// TIA Portal V17 export
// export: Created 2025-05-22T12:26:37.2129325Z, ExportSetting WithDefaults, DisplayName Totally Integrated Automation Portal, DisplayVersion V17 Update 8, DisplayName TIA Portal Openness, DisplayVersion V17 Update 8, DisplayName TIA Portal Version Control Interface, DisplayVersion V17, DisplayName SINAMICS Startdrive Advanced, DisplayVersion V17 SP2, DisplayName SINAMICS Startdrive G110M, G120, G120C, G120D, G120P, G115D, DisplayVersion V17 SP2, DisplayName SINAMICS Startdrive G130, G150, S120, S150, SINAMICS MV, S210, DisplayVersion V17 SP2, DisplayName STEP 7 Professional, DisplayVersion V17 Update 8, DisplayName SINUMERIK ONE STEP 7 Toolbox, DisplayVersion V17 Update 12, DisplayName SINUMERIK ONE PLC Basic Program Plus, DisplayVersion V17 Update 12, DisplayName SINUMERIK 840D sl STEP 7 Toolbox, DisplayVersion V17 Update 12, DisplayName STEP 7 Safety, DisplayVersion V17 Update 6, DisplayName WinCC Advanced, DisplayVersion V17 Update 8
FUNCTION_BLOCK "FB2500_FIXTURE_CLADDING"   // FB2500, LAD
{ S7_Optimized_Access := 'FALSE' }
VERSION : 0.1
// stored: AutoNumber false, IsIECCheckEnabled false, SetENOAutomatically false, UDAEnableTagReadback false
   VAR_INPUT
      PART_PRESENT_FACE_SENSOR : Bool;   // PART PRESENT FACE SENSOR
      PART_STATUS_PRESENT : Bool;   // PART STATUS PRESENT
      PART_STATUS_VIRTUAL_PART : Bool;   // PART STATUS VIRTUAL PART
      PART_STATUS_MASTER_PART : Bool;   // PART STATUS MASTER PART
      STATION_PART_PRESENT : Bool;   // STATION 1 PART PRESENT IPUT
      STATION_NO_PART : Bool;   // STATION 1 NO PART
      STATION_PART_HAT_POSITION : Bool;   // STATION 1 PART PRESENT
      STATION_PART_CLAMPED : Bool;   // STATION 1 PART CLAMPED
      STATION_PART_UNCLAMPED : Bool;   // STATION 1 PART UNCLAMPED
      STATION_CLAMPED_WITHOUT_PART : Bool;   // STATION 1 CLAMPED WITHOUT PART
      VERIFY_FIXTURE_CLAMPED : Bool;   // VERIFY FIXTURE REMAINS CLAMPED
      GRIPPER_CLOSE : Bool;   // GRIPPER CLOSE ACTION
      GRIPPER_OPEN : Bool;   // GRIPPER OPEN ACTION
      GRIPPER_CLOSED : Bool;   // GRIPPER CLOSED STATUS
      "GRIPPER OPENED" : Bool;   // GRIPPER OPENED STATUS
      M_FIXTURE_GRIPPER_CLOSE : Bool;   // M CODE FIXTURE GRIPPER CLOSE
      M_FIXTURE_GRIPPER_OPEN : Bool;   // M CODE FIXTURE GRIPPER OPEN
      UP_SEALING_STRUCTURE_CLOSED : Bool;   // UP SEALING STRUCTURE CLOSED
      DOWN_SEALING_STRUCTURE_CLOSED : Bool;   // DOWN SEALING STRUCTURE CLOSED
      PART_TYPE_FIXTURES : Bool;   // PART TYPE UNIT FIXTURES
      ROBOT_PART_LOAD_UNLOAD : Bool;   // PART LOAD/UNLOAD FROM ROBOT
      ROBOT_OUT_OF_COLLISION : Bool;   // ROBOT OUT OF COLLISION MACHINE UNIT
      E_AXIS_HOME_POS : Bool;   // E AXIS IN HOME POSITION
      W_AXIS_CLAMP_CHECK_POS : Bool;   // W AXIS IN CHECK CLAMP POSITION
      W_AXIS_UNCLAMP_CHECK_POS : Bool;   // W AXIS IN CHECK UNCLAMP POSITION
      UNIT_NO : UInt;   // UNIT NUMBER
      FIXTURE_NO : UInt;   // FIXTURE NUMBER
   END_VAR
   VAR_OUTPUT
      NOT_CLAMPED_DURING_MACHINING_A : Bool;   // NOT CLAMPED DURING MACHINING ALARM
      PART_PRESENT_DISCORDANCY_A : Bool;   // PART PRESENT DISCORDANCY ALARM
      PART_TYPE_DISCORDANCY_A : Bool;   // PART TYPE DISCORDANCY ALARM
      PART_TYPE_ORIENTATED_DISCORDANCY_A : Bool;   // PART TYPE ORIENTATED DISCORDANCY ALARM
   END_VAR
   VAR DB_SPECIFIC
      DATA : "FIXTURE_STATUS";
   END_VAR
   VAR_TEMP
      DB_NUMBER : DInt;
   END_VAR
   VAR_TEMP   // added for the SCL form of the ladder/FBD networks
      _w1 : Bool;
      _w2 : Bool;
      _w3 : Bool;
      _w4 : Bool;
      _w5 : Bool;
      _w6 : Bool;
      _w7 : Bool;
      _w8 : Bool;
      _w9 : Bool;
   END_VAR
BEGIN

NETWORK
TITLE = READ INSTANCE DB
      L     DINO;
      +     10#800000;
      T     #DB_NUMBER;


REGION Network 2: FIXTURE INPUT PART A PRESENT
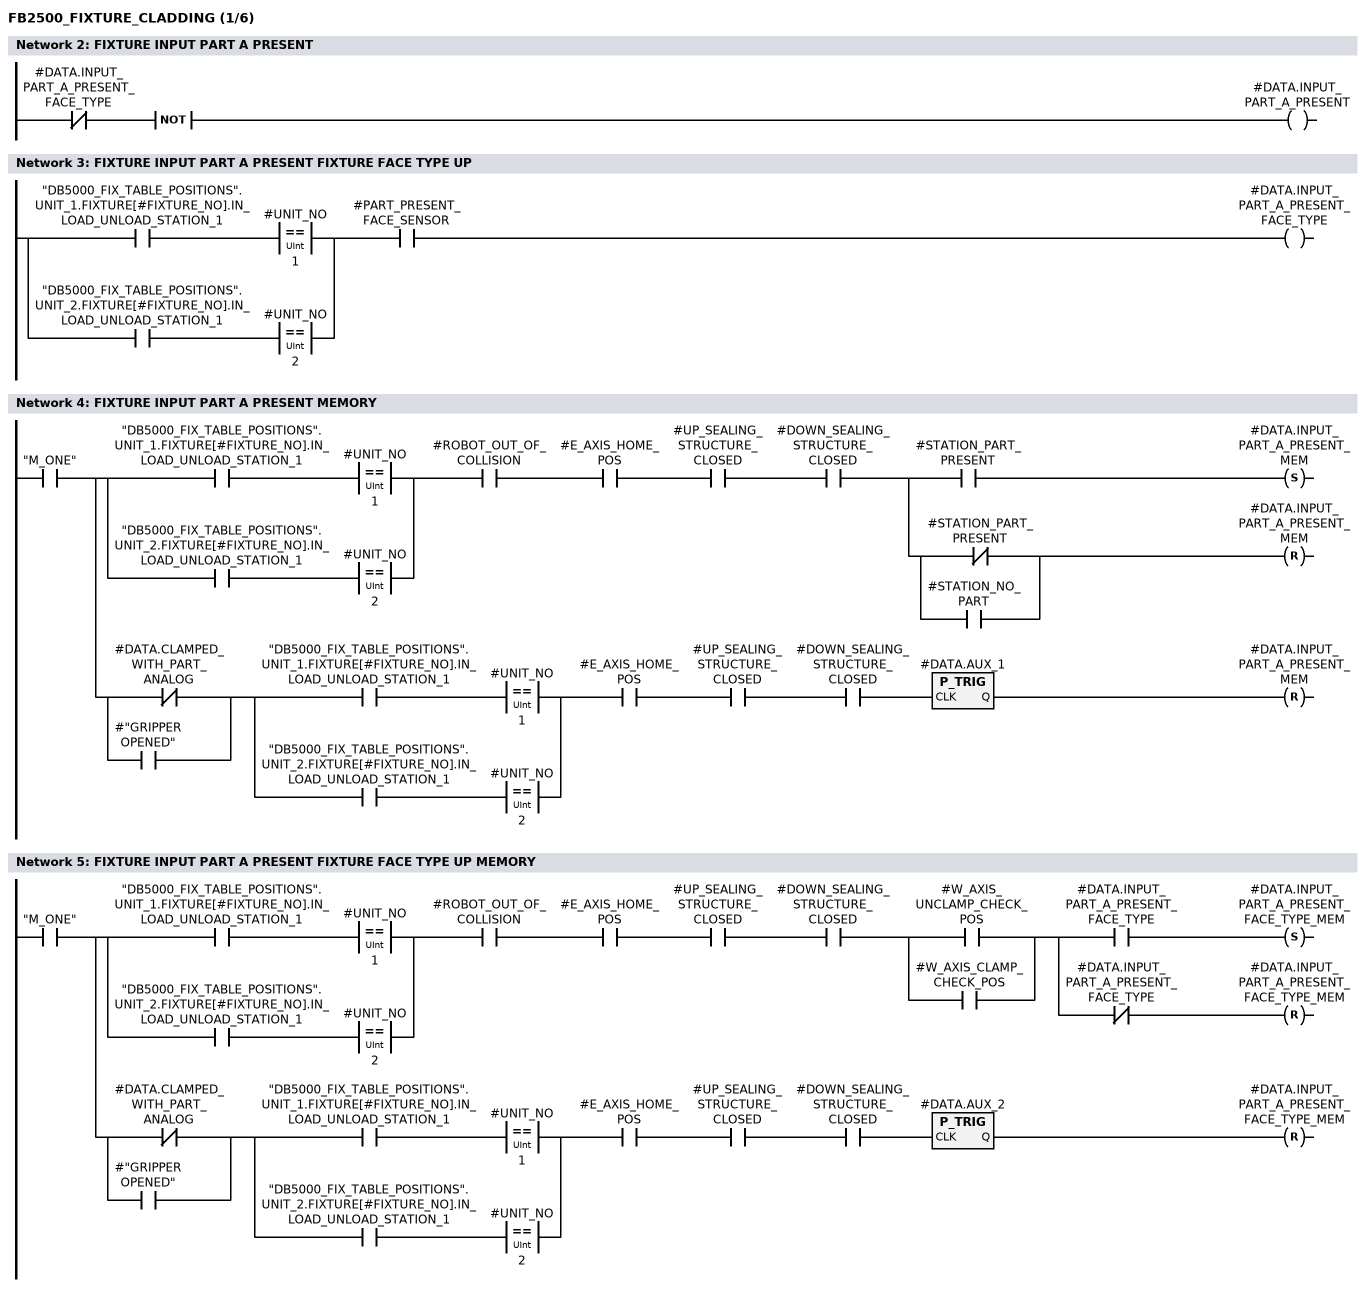
   RUNG wire#powerrail
      I_Contact( #DATA.INPUT_PART_A_PRESENT_FACE_TYPE )
      Not()
      Coil( #DATA.INPUT_PART_A_PRESENT )
   END_RUNG
   // the same network as SCL:
   #DATA.INPUT_PART_A_PRESENT := NOT (NOT #DATA.INPUT_PART_A_PRESENT_FACE_TYPE);
END_REGION

REGION Network 3: FIXTURE INPUT PART A PRESENT FIXTURE FACE TYPE UP
   RUNG wire#powerrail
      Contact( "DB5000_FIX_TABLE_POSITIONS".UNIT_1.FIXTURE[#FIXTURE_NO].IN_LOAD_UNLOAD_STATION_1 )
      { S7_Templates := "SrcType := UInt" } EQ_Contact(in1 := #UNIT_NO, in2 := 1)
      wire#w1
      Contact( #PART_PRESENT_FACE_SENSOR )
      Coil( #DATA.INPUT_PART_A_PRESENT_FACE_TYPE )
   END_RUNG
   RUNG wire#powerrail
      Contact( "DB5000_FIX_TABLE_POSITIONS".UNIT_2.FIXTURE[#FIXTURE_NO].IN_LOAD_UNLOAD_STATION_1 )
      { S7_Templates := "SrcType := UInt" } EQ_Contact(in1 := #UNIT_NO, in2 := 2)
   END_RUNG wire#w1
   // the same network as SCL:
   #DATA.INPUT_PART_A_PRESENT_FACE_TYPE := (("DB5000_FIX_TABLE_POSITIONS".UNIT_1.FIXTURE[#FIXTURE_NO].IN_LOAD_UNLOAD_STATION_1 AND (#UNIT_NO = 1)) OR ("DB5000_FIX_TABLE_POSITIONS".UNIT_2.FIXTURE[#FIXTURE_NO].IN_LOAD_UNLOAD_STATION_1 AND (#UNIT_NO = 2))) AND #PART_PRESENT_FACE_SENSOR;
END_REGION

REGION Network 4: FIXTURE INPUT PART A PRESENT MEMORY
   RUNG wire#powerrail
      Contact( "M_ONE" )
      wire#w1
      Contact( "DB5000_FIX_TABLE_POSITIONS".UNIT_1.FIXTURE[#FIXTURE_NO].IN_LOAD_UNLOAD_STATION_1 )
      { S7_Templates := "SrcType := UInt" } EQ_Contact(in1 := #UNIT_NO, in2 := 1)
      wire#w2
      Contact( #ROBOT_OUT_OF_COLLISION )
      Contact( #E_AXIS_HOME_POS )
      Contact( #UP_SEALING_STRUCTURE_CLOSED )
      Contact( #DOWN_SEALING_STRUCTURE_CLOSED )
      wire#w3
      Contact( #STATION_PART_PRESENT )
      S_Coil( #DATA.INPUT_PART_A_PRESENT_MEM )
   END_RUNG
   RUNG wire#w1
      Contact( "DB5000_FIX_TABLE_POSITIONS".UNIT_2.FIXTURE[#FIXTURE_NO].IN_LOAD_UNLOAD_STATION_1 )
      { S7_Templates := "SrcType := UInt" } EQ_Contact(in1 := #UNIT_NO, in2 := 2)
   END_RUNG wire#w2
   RUNG wire#w3
      I_Contact( #STATION_PART_PRESENT )
      wire#w4
      R_Coil( #DATA.INPUT_PART_A_PRESENT_MEM )
   END_RUNG
   RUNG wire#w3
      Contact( #STATION_NO_PART )
   END_RUNG wire#w4
   RUNG wire#w1
      I_Contact( #DATA.CLAMPED_WITH_PART_ANALOG )
      wire#w5
      Contact( "DB5000_FIX_TABLE_POSITIONS".UNIT_1.FIXTURE[#FIXTURE_NO].IN_LOAD_UNLOAD_STATION_1 )
      { S7_Templates := "SrcType := UInt" } EQ_Contact(in1 := #UNIT_NO, in2 := 1)
      wire#w6
      Contact( #E_AXIS_HOME_POS )
      Contact( #UP_SEALING_STRUCTURE_CLOSED )
      Contact( #DOWN_SEALING_STRUCTURE_CLOSED )
      P_Trig( #DATA.AUX_1 )
      R_Coil( #DATA.INPUT_PART_A_PRESENT_MEM )
   END_RUNG
   RUNG wire#w1
      Contact( #"GRIPPER OPENED" )
   END_RUNG wire#w5
   RUNG wire#w5
      Contact( "DB5000_FIX_TABLE_POSITIONS".UNIT_2.FIXTURE[#FIXTURE_NO].IN_LOAD_UNLOAD_STATION_1 )
      { S7_Templates := "SrcType := UInt" } EQ_Contact(in1 := #UNIT_NO, in2 := 2)
   END_RUNG wire#w6
   // the same network as SCL:
   #_w1 := "M_ONE" AND (("DB5000_FIX_TABLE_POSITIONS".UNIT_1.FIXTURE[#FIXTURE_NO].IN_LOAD_UNLOAD_STATION_1 AND (#UNIT_NO = 1)) OR ("DB5000_FIX_TABLE_POSITIONS".UNIT_2.FIXTURE[#FIXTURE_NO].IN_LOAD_UNLOAD_STATION_1 AND (#UNIT_NO = 2))) AND #ROBOT_OUT_OF_COLLISION AND #E_AXIS_HOME_POS AND #UP_SEALING_STRUCTURE_CLOSED AND #DOWN_SEALING_STRUCTURE_CLOSED;
   IF #_w1 AND #STATION_PART_PRESENT THEN #DATA.INPUT_PART_A_PRESENT_MEM := TRUE; END_IF;
   IF #_w1 AND (NOT #STATION_PART_PRESENT OR #STATION_NO_PART) THEN
       #DATA.INPUT_PART_A_PRESENT_MEM := FALSE;
   END_IF;
   #_w2 := "M_ONE" AND (NOT #DATA.CLAMPED_WITH_PART_ANALOG OR #"GRIPPER OPENED") AND (("DB5000_FIX_TABLE_POSITIONS".UNIT_1.FIXTURE[#FIXTURE_NO].IN_LOAD_UNLOAD_STATION_1 AND (#UNIT_NO = 1)) OR ("DB5000_FIX_TABLE_POSITIONS".UNIT_2.FIXTURE[#FIXTURE_NO].IN_LOAD_UNLOAD_STATION_1 AND (#UNIT_NO = 2))) AND #E_AXIS_HOME_POS AND #UP_SEALING_STRUCTURE_CLOSED AND #DOWN_SEALING_STRUCTURE_CLOSED;
   #_w3 := #_w2 AND NOT #DATA.AUX_1;   // rising edge
   #DATA.AUX_1 := #_w2;
   IF #_w3 THEN #DATA.INPUT_PART_A_PRESENT_MEM := FALSE; END_IF;
END_REGION

REGION Network 5: FIXTURE INPUT PART A PRESENT FIXTURE FACE TYPE UP MEMORY
   RUNG wire#powerrail
      Contact( "M_ONE" )
      wire#w1
      Contact( "DB5000_FIX_TABLE_POSITIONS".UNIT_1.FIXTURE[#FIXTURE_NO].IN_LOAD_UNLOAD_STATION_1 )
      { S7_Templates := "SrcType := UInt" } EQ_Contact(in1 := #UNIT_NO, in2 := 1)
      wire#w2
      Contact( #ROBOT_OUT_OF_COLLISION )
      Contact( #E_AXIS_HOME_POS )
      Contact( #UP_SEALING_STRUCTURE_CLOSED )
      Contact( #DOWN_SEALING_STRUCTURE_CLOSED )
      wire#w3
      Contact( #W_AXIS_UNCLAMP_CHECK_POS )
      wire#w4
      Contact( #DATA.INPUT_PART_A_PRESENT_FACE_TYPE )
      S_Coil( #DATA.INPUT_PART_A_PRESENT_FACE_TYPE_MEM )
   END_RUNG
   RUNG wire#w1
      Contact( "DB5000_FIX_TABLE_POSITIONS".UNIT_2.FIXTURE[#FIXTURE_NO].IN_LOAD_UNLOAD_STATION_1 )
      { S7_Templates := "SrcType := UInt" } EQ_Contact(in1 := #UNIT_NO, in2 := 2)
   END_RUNG wire#w2
   RUNG wire#w3
      Contact( #W_AXIS_CLAMP_CHECK_POS )
   END_RUNG wire#w4
   RUNG wire#w4
      I_Contact( #DATA.INPUT_PART_A_PRESENT_FACE_TYPE )
      R_Coil( #DATA.INPUT_PART_A_PRESENT_FACE_TYPE_MEM )
   END_RUNG
   RUNG wire#w1
      I_Contact( #DATA.CLAMPED_WITH_PART_ANALOG )
      wire#w5
      Contact( "DB5000_FIX_TABLE_POSITIONS".UNIT_1.FIXTURE[#FIXTURE_NO].IN_LOAD_UNLOAD_STATION_1 )
      { S7_Templates := "SrcType := UInt" } EQ_Contact(in1 := #UNIT_NO, in2 := 1)
      wire#w6
      Contact( #E_AXIS_HOME_POS )
      Contact( #UP_SEALING_STRUCTURE_CLOSED )
      Contact( #DOWN_SEALING_STRUCTURE_CLOSED )
      P_Trig( #DATA.AUX_2 )
      R_Coil( #DATA.INPUT_PART_A_PRESENT_FACE_TYPE_MEM )
   END_RUNG
   RUNG wire#w1
      Contact( #"GRIPPER OPENED" )
   END_RUNG wire#w5
   RUNG wire#w5
      Contact( "DB5000_FIX_TABLE_POSITIONS".UNIT_2.FIXTURE[#FIXTURE_NO].IN_LOAD_UNLOAD_STATION_1 )
      { S7_Templates := "SrcType := UInt" } EQ_Contact(in1 := #UNIT_NO, in2 := 2)
   END_RUNG wire#w6
   // the same network as SCL:
   #_w1 := "M_ONE" AND (("DB5000_FIX_TABLE_POSITIONS".UNIT_1.FIXTURE[#FIXTURE_NO].IN_LOAD_UNLOAD_STATION_1 AND (#UNIT_NO = 1)) OR ("DB5000_FIX_TABLE_POSITIONS".UNIT_2.FIXTURE[#FIXTURE_NO].IN_LOAD_UNLOAD_STATION_1 AND (#UNIT_NO = 2))) AND #ROBOT_OUT_OF_COLLISION AND #E_AXIS_HOME_POS AND #UP_SEALING_STRUCTURE_CLOSED AND #DOWN_SEALING_STRUCTURE_CLOSED AND (#W_AXIS_UNCLAMP_CHECK_POS OR #W_AXIS_CLAMP_CHECK_POS);
   IF #_w1 AND #DATA.INPUT_PART_A_PRESENT_FACE_TYPE THEN
       #DATA.INPUT_PART_A_PRESENT_FACE_TYPE_MEM := TRUE;
   END_IF;
   IF #_w1 AND NOT #DATA.INPUT_PART_A_PRESENT_FACE_TYPE THEN
       #DATA.INPUT_PART_A_PRESENT_FACE_TYPE_MEM := FALSE;
   END_IF;
   #_w2 := "M_ONE" AND (NOT #DATA.CLAMPED_WITH_PART_ANALOG OR #"GRIPPER OPENED") AND (("DB5000_FIX_TABLE_POSITIONS".UNIT_1.FIXTURE[#FIXTURE_NO].IN_LOAD_UNLOAD_STATION_1 AND (#UNIT_NO = 1)) OR ("DB5000_FIX_TABLE_POSITIONS".UNIT_2.FIXTURE[#FIXTURE_NO].IN_LOAD_UNLOAD_STATION_1 AND (#UNIT_NO = 2))) AND #E_AXIS_HOME_POS AND #UP_SEALING_STRUCTURE_CLOSED AND #DOWN_SEALING_STRUCTURE_CLOSED;
   #_w3 := #_w2 AND NOT #DATA.AUX_2;   // rising edge
   #DATA.AUX_2 := #_w2;
   IF #_w3 THEN #DATA.INPUT_PART_A_PRESENT_FACE_TYPE_MEM := FALSE; END_IF;
END_REGION

REGION Network 6: ANY PART PRESENT
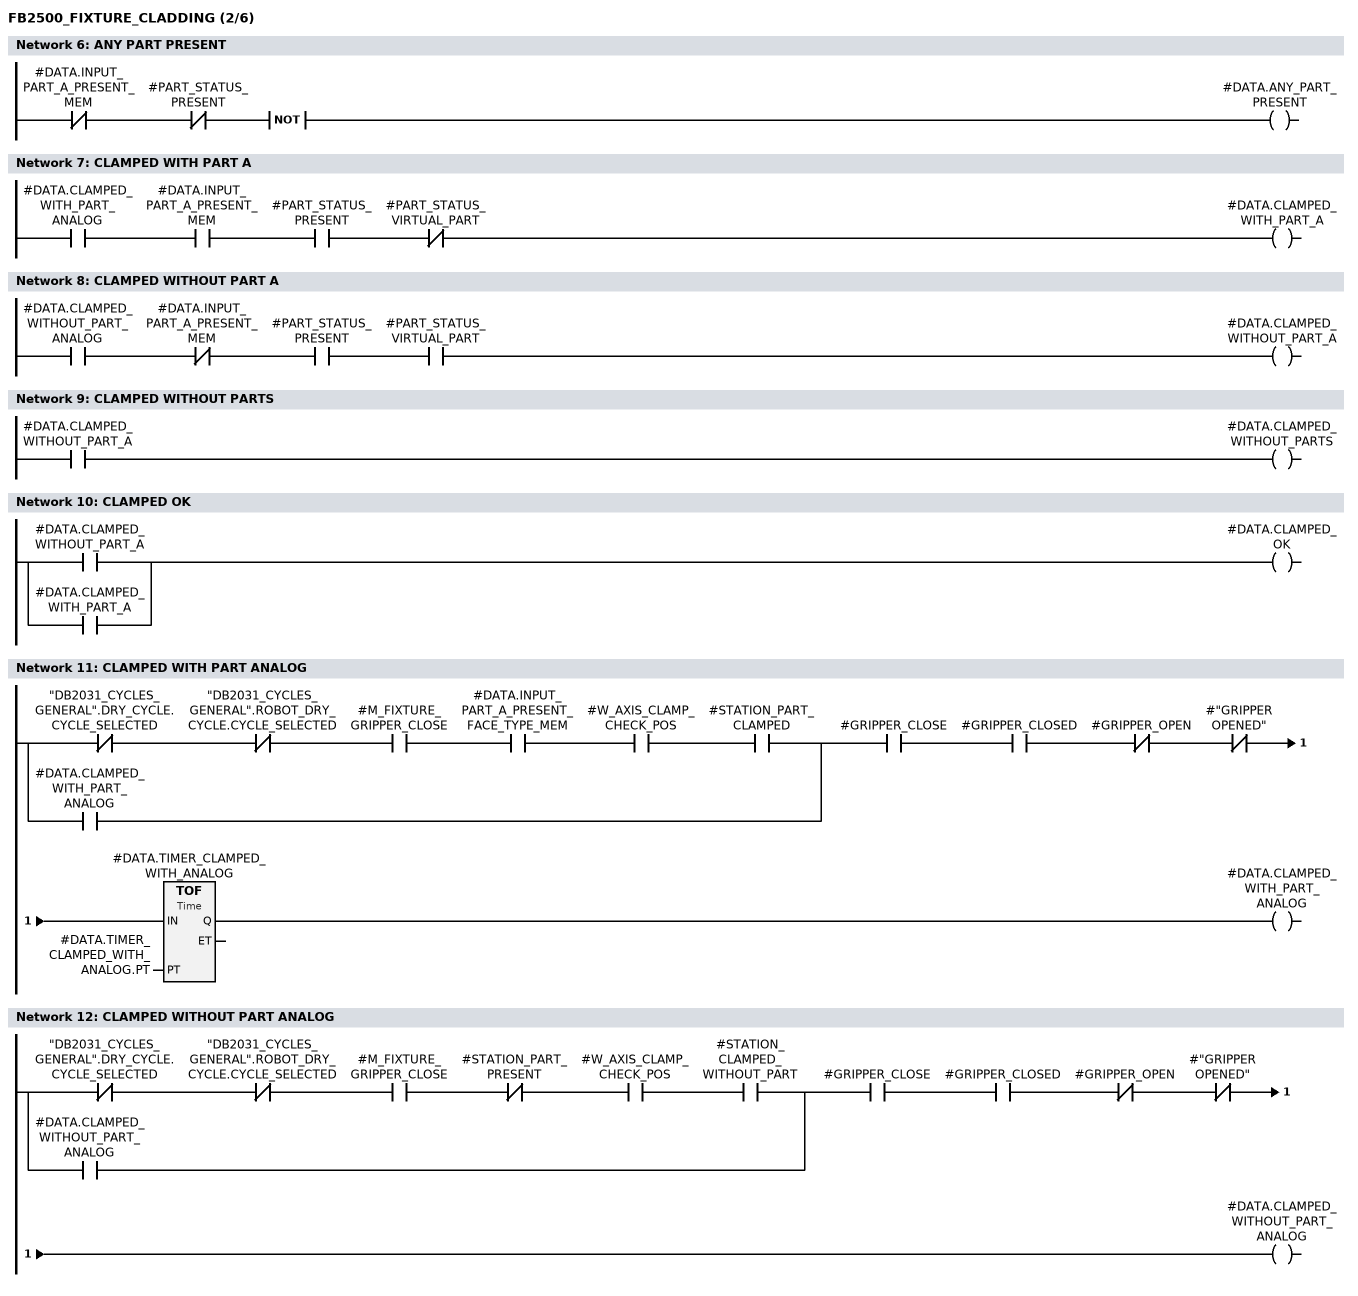
   RUNG wire#powerrail
      I_Contact( #DATA.INPUT_PART_A_PRESENT_MEM )
      I_Contact( #PART_STATUS_PRESENT )
      Not()
      Coil( #DATA.ANY_PART_PRESENT )
   END_RUNG
   // the same network as SCL:
   #DATA.ANY_PART_PRESENT := NOT (NOT #DATA.INPUT_PART_A_PRESENT_MEM AND NOT #PART_STATUS_PRESENT);
END_REGION

REGION Network 7: CLAMPED WITH PART A
   RUNG wire#powerrail
      Contact( #DATA.CLAMPED_WITH_PART_ANALOG )
      Contact( #DATA.INPUT_PART_A_PRESENT_MEM )
      Contact( #PART_STATUS_PRESENT )
      I_Contact( #PART_STATUS_VIRTUAL_PART )
      Coil( #DATA.CLAMPED_WITH_PART_A )
   END_RUNG
   // the same network as SCL:
   #DATA.CLAMPED_WITH_PART_A := #DATA.CLAMPED_WITH_PART_ANALOG AND #DATA.INPUT_PART_A_PRESENT_MEM AND #PART_STATUS_PRESENT AND NOT #PART_STATUS_VIRTUAL_PART;
END_REGION

REGION Network 8: CLAMPED WITHOUT PART A
   RUNG wire#powerrail
      Contact( #DATA.CLAMPED_WITHOUT_PART_ANALOG )
      I_Contact( #DATA.INPUT_PART_A_PRESENT_MEM )
      Contact( #PART_STATUS_PRESENT )
      Contact( #PART_STATUS_VIRTUAL_PART )
      Coil( #DATA.CLAMPED_WITHOUT_PART_A )
   END_RUNG
   // the same network as SCL:
   #DATA.CLAMPED_WITHOUT_PART_A := #DATA.CLAMPED_WITHOUT_PART_ANALOG AND NOT #DATA.INPUT_PART_A_PRESENT_MEM AND #PART_STATUS_PRESENT AND #PART_STATUS_VIRTUAL_PART;
END_REGION

REGION Network 9: CLAMPED WITHOUT PARTS
   RUNG wire#powerrail
      Contact( #DATA.CLAMPED_WITHOUT_PART_A )
      Coil( #DATA.CLAMPED_WITHOUT_PARTS )
   END_RUNG
   // the same network as SCL:
   #DATA.CLAMPED_WITHOUT_PARTS := #DATA.CLAMPED_WITHOUT_PART_A;
END_REGION

REGION Network 10: CLAMPED OK
   RUNG wire#powerrail
      Contact( #DATA.CLAMPED_WITHOUT_PART_A )
      wire#w1
      Coil( #DATA.CLAMPED_OK )
   END_RUNG
   RUNG wire#powerrail
      Contact( #DATA.CLAMPED_WITH_PART_A )
   END_RUNG wire#w1
   // the same network as SCL:
   #DATA.CLAMPED_OK := #DATA.CLAMPED_WITHOUT_PART_A OR #DATA.CLAMPED_WITH_PART_A;
END_REGION

REGION Network 11: CLAMPED WITH PART ANALOG
   RUNG wire#powerrail
      I_Contact( "DB2031_CYCLES_GENERAL".DRY_CYCLE.CYCLE_SELECTED )
      I_Contact( "DB2031_CYCLES_GENERAL".ROBOT_DRY_CYCLE.CYCLE_SELECTED )
      Contact( #M_FIXTURE_GRIPPER_CLOSE )
      Contact( #DATA.INPUT_PART_A_PRESENT_FACE_TYPE_MEM )
      Contact( #W_AXIS_CLAMP_CHECK_POS )
      Contact( #STATION_PART_CLAMPED )
      wire#w1
      Contact( #GRIPPER_CLOSE )
      Contact( #GRIPPER_CLOSED )
      I_Contact( #GRIPPER_OPEN )
      I_Contact( #"GRIPPER OPENED" )
      { S7_Templates := "time_type := Time" } #DATA.TIMER_CLAMPED_WITH_ANALOG.TOF(pt := #DATA.TIMER_CLAMPED_WITH_ANALOG.PT, et =>)
      Coil( #DATA.CLAMPED_WITH_PART_ANALOG )
   END_RUNG
   RUNG wire#powerrail
      Contact( #DATA.CLAMPED_WITH_PART_ANALOG )
   END_RUNG wire#w1
   // the same network as SCL:
   #DATA.TIMER_CLAMPED_WITH_ANALOG.TOF(IN := ((NOT "DB2031_CYCLES_GENERAL".DRY_CYCLE.CYCLE_SELECTED AND NOT "DB2031_CYCLES_GENERAL".ROBOT_DRY_CYCLE.CYCLE_SELECTED AND #M_FIXTURE_GRIPPER_CLOSE AND #DATA.INPUT_PART_A_PRESENT_FACE_TYPE_MEM AND #W_AXIS_CLAMP_CHECK_POS AND #STATION_PART_CLAMPED) OR #DATA.CLAMPED_WITH_PART_ANALOG) AND #GRIPPER_CLOSE AND #GRIPPER_CLOSED AND NOT #GRIPPER_OPEN AND NOT #"GRIPPER OPENED",
                           PT := #DATA.TIMER_CLAMPED_WITH_ANALOG.PT);
   #DATA.CLAMPED_WITH_PART_ANALOG := #DATA.TIMER_CLAMPED_WITH_ANALOG.Q;
END_REGION

REGION Network 12: CLAMPED WITHOUT PART ANALOG
   RUNG wire#powerrail
      I_Contact( "DB2031_CYCLES_GENERAL".DRY_CYCLE.CYCLE_SELECTED )
      I_Contact( "DB2031_CYCLES_GENERAL".ROBOT_DRY_CYCLE.CYCLE_SELECTED )
      Contact( #M_FIXTURE_GRIPPER_CLOSE )
      I_Contact( #STATION_PART_PRESENT )
      Contact( #W_AXIS_CLAMP_CHECK_POS )
      Contact( #STATION_CLAMPED_WITHOUT_PART )
      wire#w1
      Contact( #GRIPPER_CLOSE )
      Contact( #GRIPPER_CLOSED )
      I_Contact( #GRIPPER_OPEN )
      I_Contact( #"GRIPPER OPENED" )
      Coil( #DATA.CLAMPED_WITHOUT_PART_ANALOG )
   END_RUNG
   RUNG wire#powerrail
      Contact( #DATA.CLAMPED_WITHOUT_PART_ANALOG )
   END_RUNG wire#w1
   // the same network as SCL:
   #DATA.CLAMPED_WITHOUT_PART_ANALOG := ((NOT "DB2031_CYCLES_GENERAL".DRY_CYCLE.CYCLE_SELECTED AND NOT "DB2031_CYCLES_GENERAL".ROBOT_DRY_CYCLE.CYCLE_SELECTED AND #M_FIXTURE_GRIPPER_CLOSE AND NOT #STATION_PART_PRESENT AND #W_AXIS_CLAMP_CHECK_POS AND #STATION_CLAMPED_WITHOUT_PART) OR #DATA.CLAMPED_WITHOUT_PART_ANALOG) AND #GRIPPER_CLOSE AND #GRIPPER_CLOSED AND NOT #GRIPPER_OPEN AND NOT #"GRIPPER OPENED";
END_REGION

REGION Network 13: UNCLAMPED ANALOG
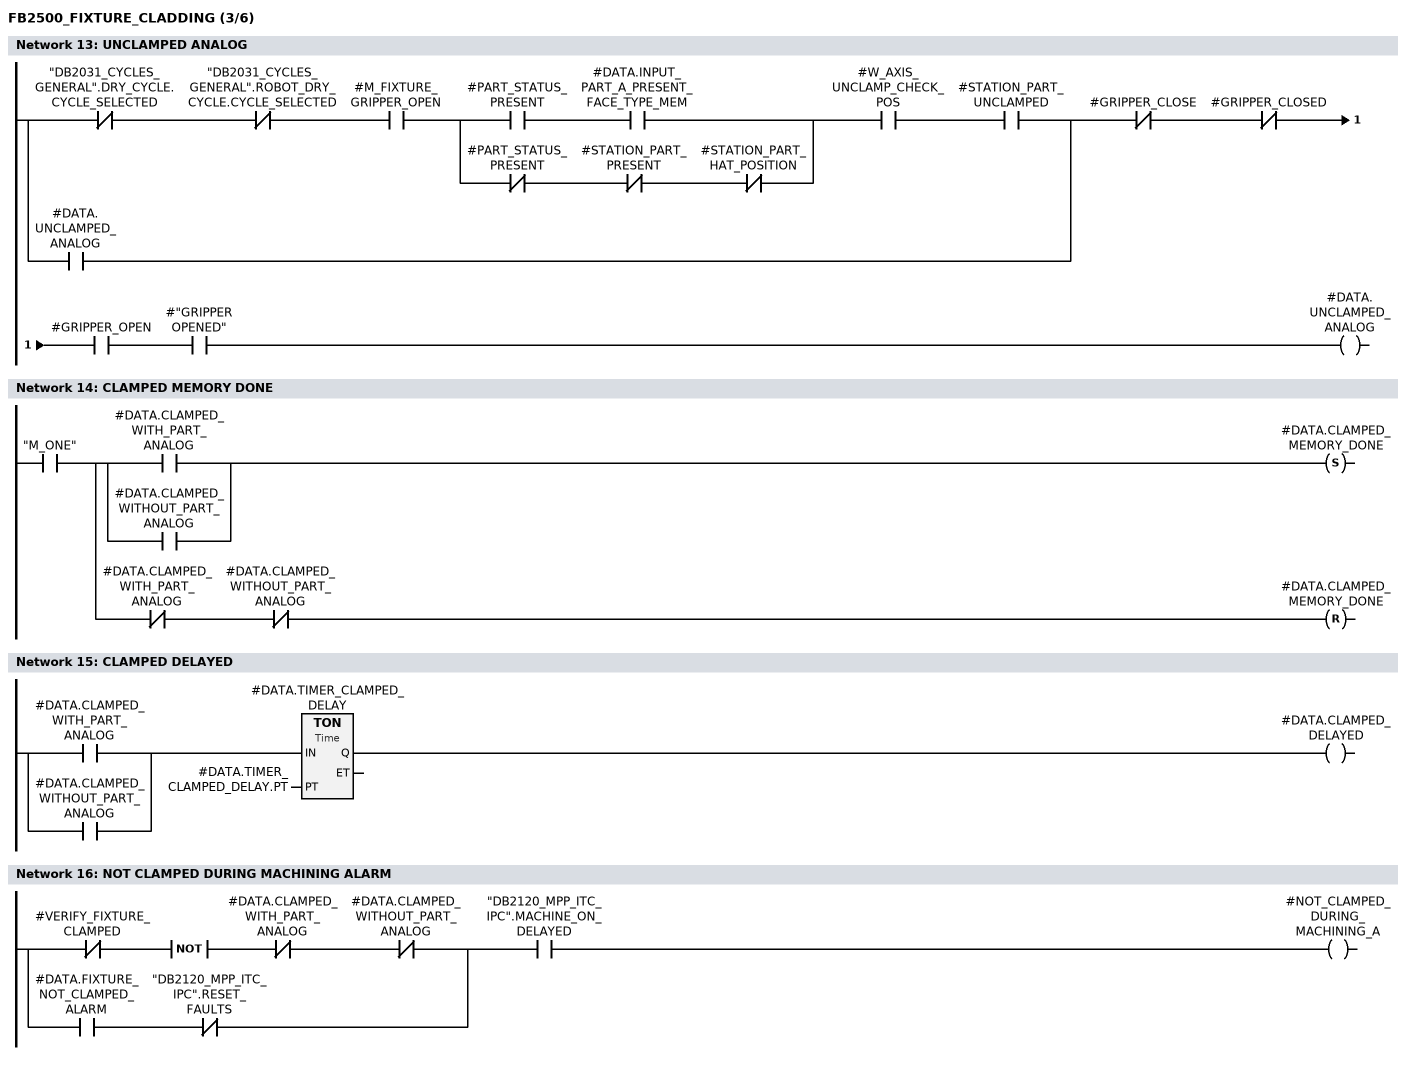
   RUNG wire#powerrail
      I_Contact( "DB2031_CYCLES_GENERAL".DRY_CYCLE.CYCLE_SELECTED )
      I_Contact( "DB2031_CYCLES_GENERAL".ROBOT_DRY_CYCLE.CYCLE_SELECTED )
      Contact( #M_FIXTURE_GRIPPER_OPEN )
      wire#w1
      Contact( #PART_STATUS_PRESENT )
      Contact( #DATA.INPUT_PART_A_PRESENT_FACE_TYPE_MEM )
      wire#w2
      Contact( #W_AXIS_UNCLAMP_CHECK_POS )
      Contact( #STATION_PART_UNCLAMPED )
      wire#w3
      I_Contact( #GRIPPER_CLOSE )
      I_Contact( #GRIPPER_CLOSED )
      Contact( #GRIPPER_OPEN )
      Contact( #"GRIPPER OPENED" )
      Coil( #DATA.UNCLAMPED_ANALOG )
   END_RUNG
   RUNG wire#w1
      I_Contact( #PART_STATUS_PRESENT )
      I_Contact( #STATION_PART_PRESENT )
      I_Contact( #STATION_PART_HAT_POSITION )
   END_RUNG wire#w2
   RUNG wire#powerrail
      Contact( #DATA.UNCLAMPED_ANALOG )
   END_RUNG wire#w3
   // the same network as SCL:
   #DATA.UNCLAMPED_ANALOG := ((NOT "DB2031_CYCLES_GENERAL".DRY_CYCLE.CYCLE_SELECTED AND NOT "DB2031_CYCLES_GENERAL".ROBOT_DRY_CYCLE.CYCLE_SELECTED AND #M_FIXTURE_GRIPPER_OPEN AND ((#PART_STATUS_PRESENT AND #DATA.INPUT_PART_A_PRESENT_FACE_TYPE_MEM) OR (NOT #PART_STATUS_PRESENT AND NOT #STATION_PART_PRESENT AND NOT #STATION_PART_HAT_POSITION)) AND #W_AXIS_UNCLAMP_CHECK_POS AND #STATION_PART_UNCLAMPED) OR #DATA.UNCLAMPED_ANALOG) AND NOT #GRIPPER_CLOSE AND NOT #GRIPPER_CLOSED AND #GRIPPER_OPEN AND #"GRIPPER OPENED";
END_REGION

REGION Network 14: CLAMPED MEMORY DONE
   RUNG wire#powerrail
      Contact( "M_ONE" )
      wire#w1
      Contact( #DATA.CLAMPED_WITH_PART_ANALOG )
      wire#w2
      S_Coil( #DATA.CLAMPED_MEMORY_DONE )
   END_RUNG
   RUNG wire#w1
      Contact( #DATA.CLAMPED_WITHOUT_PART_ANALOG )
   END_RUNG wire#w2
   RUNG wire#w1
      I_Contact( #DATA.CLAMPED_WITH_PART_ANALOG )
      I_Contact( #DATA.CLAMPED_WITHOUT_PART_ANALOG )
      R_Coil( #DATA.CLAMPED_MEMORY_DONE )
   END_RUNG
   // the same network as SCL:
   IF "M_ONE" AND (#DATA.CLAMPED_WITH_PART_ANALOG OR #DATA.CLAMPED_WITHOUT_PART_ANALOG) THEN
       #DATA.CLAMPED_MEMORY_DONE := TRUE;
   END_IF;
   IF "M_ONE" AND NOT #DATA.CLAMPED_WITH_PART_ANALOG AND NOT #DATA.CLAMPED_WITHOUT_PART_ANALOG THEN
       #DATA.CLAMPED_MEMORY_DONE := FALSE;
   END_IF;
END_REGION

REGION Network 15: CLAMPED DELAYED
   RUNG wire#powerrail
      Contact( #DATA.CLAMPED_WITH_PART_ANALOG )
      wire#w1
      { S7_Templates := "time_type := Time" } #DATA.TIMER_CLAMPED_DELAY.TON(pt := #DATA.TIMER_CLAMPED_DELAY.PT, et =>)
      Coil( #DATA.CLAMPED_DELAYED )
   END_RUNG
   RUNG wire#powerrail
      Contact( #DATA.CLAMPED_WITHOUT_PART_ANALOG )
   END_RUNG wire#w1
   // the same network as SCL:
   #DATA.TIMER_CLAMPED_DELAY.TON(IN := #DATA.CLAMPED_WITH_PART_ANALOG OR #DATA.CLAMPED_WITHOUT_PART_ANALOG,
                           PT := #DATA.TIMER_CLAMPED_DELAY.PT);
   #DATA.CLAMPED_DELAYED := #DATA.TIMER_CLAMPED_DELAY.Q;
END_REGION

REGION Network 16: NOT CLAMPED DURING MACHINING ALARM
   RUNG wire#powerrail
      I_Contact( #VERIFY_FIXTURE_CLAMPED )
      Not()
      I_Contact( #DATA.CLAMPED_WITH_PART_ANALOG )
      I_Contact( #DATA.CLAMPED_WITHOUT_PART_ANALOG )
      wire#w1
      Contact( "DB2120_MPP_ITC_IPC".MACHINE_ON_DELAYED )
      Coil( #NOT_CLAMPED_DURING_MACHINING_A )
   END_RUNG
   RUNG wire#powerrail
      Contact( #DATA.FIXTURE_NOT_CLAMPED_ALARM )
      I_Contact( "DB2120_MPP_ITC_IPC".RESET_FAULTS )
   END_RUNG wire#w1
   // the same network as SCL:
   #NOT_CLAMPED_DURING_MACHINING_A := ((NOT (NOT #VERIFY_FIXTURE_CLAMPED) AND NOT #DATA.CLAMPED_WITH_PART_ANALOG AND NOT #DATA.CLAMPED_WITHOUT_PART_ANALOG) OR (#DATA.FIXTURE_NOT_CLAMPED_ALARM AND NOT "DB2120_MPP_ITC_IPC".RESET_FAULTS)) AND "DB2120_MPP_ITC_IPC".MACHINE_ON_DELAYED;
END_REGION

REGION Network 17: PART A PRESENT DISCORDANCY ALARM
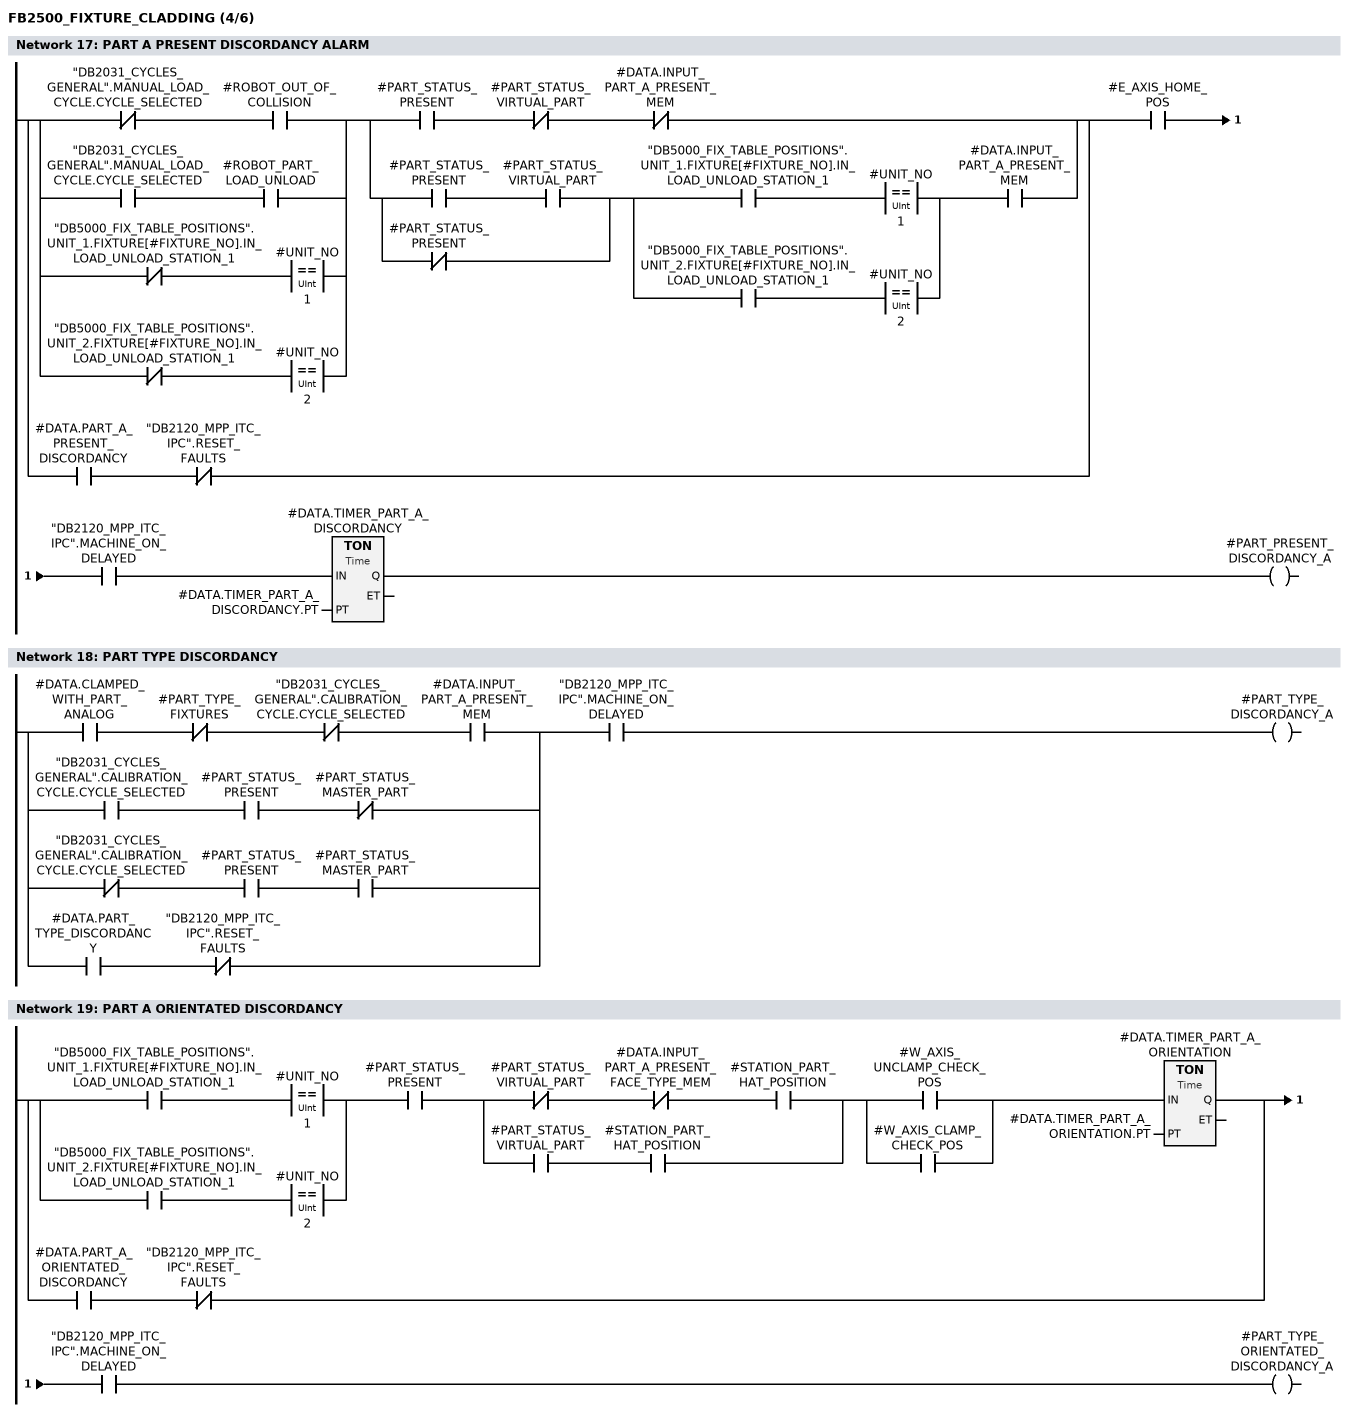
   RUNG wire#powerrail
      I_Contact( "DB2031_CYCLES_GENERAL".MANUAL_LOAD_CYCLE.CYCLE_SELECTED )
      Contact( #ROBOT_OUT_OF_COLLISION )
      wire#w1
      Contact( #PART_STATUS_PRESENT )
      I_Contact( #PART_STATUS_VIRTUAL_PART )
      I_Contact( #DATA.INPUT_PART_A_PRESENT_MEM )
      wire#w2
      Contact( #E_AXIS_HOME_POS )
      Contact( "DB2120_MPP_ITC_IPC".MACHINE_ON_DELAYED )
      { S7_Templates := "time_type := Time" } #DATA.TIMER_PART_A_DISCORDANCY.TON(pt := #DATA.TIMER_PART_A_DISCORDANCY.PT, et =>)
      Coil( #PART_PRESENT_DISCORDANCY_A )
   END_RUNG
   RUNG wire#powerrail
      Contact( "DB2031_CYCLES_GENERAL".MANUAL_LOAD_CYCLE.CYCLE_SELECTED )
      Contact( #ROBOT_PART_LOAD_UNLOAD )
   END_RUNG wire#w1
   RUNG wire#powerrail
      I_Contact( "DB5000_FIX_TABLE_POSITIONS".UNIT_1.FIXTURE[#FIXTURE_NO].IN_LOAD_UNLOAD_STATION_1 )
      { S7_Templates := "SrcType := UInt" } EQ_Contact(in1 := #UNIT_NO, in2 := 1)
   END_RUNG wire#w1
   RUNG wire#powerrail
      I_Contact( "DB5000_FIX_TABLE_POSITIONS".UNIT_2.FIXTURE[#FIXTURE_NO].IN_LOAD_UNLOAD_STATION_1 )
      { S7_Templates := "SrcType := UInt" } EQ_Contact(in1 := #UNIT_NO, in2 := 2)
   END_RUNG wire#w1
   RUNG wire#w1
      Contact( #PART_STATUS_PRESENT )
      Contact( #PART_STATUS_VIRTUAL_PART )
      wire#w3
      Contact( "DB5000_FIX_TABLE_POSITIONS".UNIT_1.FIXTURE[#FIXTURE_NO].IN_LOAD_UNLOAD_STATION_1 )
      { S7_Templates := "SrcType := UInt" } EQ_Contact(in1 := #UNIT_NO, in2 := 1)
      wire#w4
      Contact( #DATA.INPUT_PART_A_PRESENT_MEM )
   END_RUNG wire#w2
   RUNG wire#w1
      I_Contact( #PART_STATUS_PRESENT )
   END_RUNG wire#w3
   RUNG wire#w3
      Contact( "DB5000_FIX_TABLE_POSITIONS".UNIT_2.FIXTURE[#FIXTURE_NO].IN_LOAD_UNLOAD_STATION_1 )
      { S7_Templates := "SrcType := UInt" } EQ_Contact(in1 := #UNIT_NO, in2 := 2)
   END_RUNG wire#w4
   RUNG wire#powerrail
      Contact( #DATA.PART_A_PRESENT_DISCORDANCY )
      I_Contact( "DB2120_MPP_ITC_IPC".RESET_FAULTS )
   END_RUNG wire#w2
   // the same network as SCL:
   #DATA.TIMER_PART_A_DISCORDANCY.TON(IN := ((((NOT "DB2031_CYCLES_GENERAL".MANUAL_LOAD_CYCLE.CYCLE_SELECTED AND #ROBOT_OUT_OF_COLLISION) OR ("DB2031_CYCLES_GENERAL".MANUAL_LOAD_CYCLE.CYCLE_SELECTED AND #ROBOT_PART_LOAD_UNLOAD) OR (NOT "DB5000_FIX_TABLE_POSITIONS".UNIT_1.FIXTURE[#FIXTURE_NO].IN_LOAD_UNLOAD_STATION_1 AND (#UNIT_NO = 1)) OR (NOT "DB5000_FIX_TABLE_POSITIONS".UNIT_2.FIXTURE[#FIXTURE_NO].IN_LOAD_UNLOAD_STATION_1 AND (#UNIT_NO = 2))) AND ((#PART_STATUS_PRESENT AND NOT #PART_STATUS_VIRTUAL_PART AND NOT #DATA.INPUT_PART_A_PRESENT_MEM) OR (((#PART_STATUS_PRESENT AND #PART_STATUS_VIRTUAL_PART) OR NOT #PART_STATUS_PRESENT) AND (("DB5000_FIX_TABLE_POSITIONS".UNIT_1.FIXTURE[#FIXTURE_NO].IN_LOAD_UNLOAD_STATION_1 AND (#UNIT_NO = 1)) OR ("DB5000_FIX_TABLE_POSITIONS".UNIT_2.FIXTURE[#FIXTURE_NO].IN_LOAD_UNLOAD_STATION_1 AND (#UNIT_NO = 2))) AND #DATA.INPUT_PART_A_PRESENT_MEM))) OR (#DATA.PART_A_PRESENT_DISCORDANCY AND NOT "DB2120_MPP_ITC_IPC".RESET_FAULTS)) AND #E_AXIS_HOME_POS AND "DB2120_MPP_ITC_IPC".MACHINE_ON_DELAYED,
                           PT := #DATA.TIMER_PART_A_DISCORDANCY.PT);
   #PART_PRESENT_DISCORDANCY_A := #DATA.TIMER_PART_A_DISCORDANCY.Q;
END_REGION

REGION Network 18: PART TYPE DISCORDANCY
   RUNG wire#powerrail
      Contact( #DATA.CLAMPED_WITH_PART_ANALOG )
      I_Contact( #PART_TYPE_FIXTURES )
      I_Contact( "DB2031_CYCLES_GENERAL".CALIBRATION_CYCLE.CYCLE_SELECTED )
      Contact( #DATA.INPUT_PART_A_PRESENT_MEM )
      wire#w1
      Contact( "DB2120_MPP_ITC_IPC".MACHINE_ON_DELAYED )
      Coil( #PART_TYPE_DISCORDANCY_A )
   END_RUNG
   RUNG wire#powerrail
      Contact( "DB2031_CYCLES_GENERAL".CALIBRATION_CYCLE.CYCLE_SELECTED )
      Contact( #PART_STATUS_PRESENT )
      I_Contact( #PART_STATUS_MASTER_PART )
   END_RUNG wire#w1
   RUNG wire#powerrail
      I_Contact( "DB2031_CYCLES_GENERAL".CALIBRATION_CYCLE.CYCLE_SELECTED )
      Contact( #PART_STATUS_PRESENT )
      Contact( #PART_STATUS_MASTER_PART )
   END_RUNG wire#w1
   RUNG wire#powerrail
      Contact( #DATA.PART_TYPE_DISCORDANCY )
      I_Contact( "DB2120_MPP_ITC_IPC".RESET_FAULTS )
   END_RUNG wire#w1
   // the same network as SCL:
   #PART_TYPE_DISCORDANCY_A := ((#DATA.CLAMPED_WITH_PART_ANALOG AND NOT #PART_TYPE_FIXTURES AND NOT "DB2031_CYCLES_GENERAL".CALIBRATION_CYCLE.CYCLE_SELECTED AND #DATA.INPUT_PART_A_PRESENT_MEM) OR ("DB2031_CYCLES_GENERAL".CALIBRATION_CYCLE.CYCLE_SELECTED AND #PART_STATUS_PRESENT AND NOT #PART_STATUS_MASTER_PART) OR (NOT "DB2031_CYCLES_GENERAL".CALIBRATION_CYCLE.CYCLE_SELECTED AND #PART_STATUS_PRESENT AND #PART_STATUS_MASTER_PART) OR (#DATA.PART_TYPE_DISCORDANCY AND NOT "DB2120_MPP_ITC_IPC".RESET_FAULTS)) AND "DB2120_MPP_ITC_IPC".MACHINE_ON_DELAYED;
END_REGION

REGION Network 19: PART A ORIENTATED DISCORDANCY
   RUNG wire#powerrail
      Contact( "DB5000_FIX_TABLE_POSITIONS".UNIT_1.FIXTURE[#FIXTURE_NO].IN_LOAD_UNLOAD_STATION_1 )
      { S7_Templates := "SrcType := UInt" } EQ_Contact(in1 := #UNIT_NO, in2 := 1)
      wire#w1
      Contact( #PART_STATUS_PRESENT )
      wire#w2
      I_Contact( #PART_STATUS_VIRTUAL_PART )
      I_Contact( #DATA.INPUT_PART_A_PRESENT_FACE_TYPE_MEM )
      Contact( #STATION_PART_HAT_POSITION )
      wire#w3
      Contact( #W_AXIS_UNCLAMP_CHECK_POS )
      wire#w4
      { S7_Templates := "time_type := Time" } #DATA.TIMER_PART_A_ORIENTATION.TON(pt := #DATA.TIMER_PART_A_ORIENTATION.PT, et =>)
      wire#w5
      Contact( "DB2120_MPP_ITC_IPC".MACHINE_ON_DELAYED )
      Coil( #PART_TYPE_ORIENTATED_DISCORDANCY_A )
   END_RUNG
   RUNG wire#powerrail
      Contact( "DB5000_FIX_TABLE_POSITIONS".UNIT_2.FIXTURE[#FIXTURE_NO].IN_LOAD_UNLOAD_STATION_1 )
      { S7_Templates := "SrcType := UInt" } EQ_Contact(in1 := #UNIT_NO, in2 := 2)
   END_RUNG wire#w1
   RUNG wire#w2
      Contact( #PART_STATUS_VIRTUAL_PART )
      Contact( #STATION_PART_HAT_POSITION )
   END_RUNG wire#w3
   RUNG wire#w3
      Contact( #W_AXIS_CLAMP_CHECK_POS )
   END_RUNG wire#w4
   RUNG wire#powerrail
      Contact( #DATA.PART_A_ORIENTATED_DISCORDANCY )
      I_Contact( "DB2120_MPP_ITC_IPC".RESET_FAULTS )
   END_RUNG wire#w5
   // the same network as SCL:
   #DATA.TIMER_PART_A_ORIENTATION.TON(IN := (("DB5000_FIX_TABLE_POSITIONS".UNIT_1.FIXTURE[#FIXTURE_NO].IN_LOAD_UNLOAD_STATION_1 AND (#UNIT_NO = 1)) OR ("DB5000_FIX_TABLE_POSITIONS".UNIT_2.FIXTURE[#FIXTURE_NO].IN_LOAD_UNLOAD_STATION_1 AND (#UNIT_NO = 2))) AND #PART_STATUS_PRESENT AND ((NOT #PART_STATUS_VIRTUAL_PART AND NOT #DATA.INPUT_PART_A_PRESENT_FACE_TYPE_MEM AND #STATION_PART_HAT_POSITION) OR (#PART_STATUS_VIRTUAL_PART AND #STATION_PART_HAT_POSITION)) AND (#W_AXIS_UNCLAMP_CHECK_POS OR #W_AXIS_CLAMP_CHECK_POS),
                           PT := #DATA.TIMER_PART_A_ORIENTATION.PT);
   #PART_TYPE_ORIENTATED_DISCORDANCY_A := (#DATA.TIMER_PART_A_ORIENTATION.Q OR (#DATA.PART_A_ORIENTATED_DISCORDANCY AND NOT "DB2120_MPP_ITC_IPC".RESET_FAULTS)) AND "DB2120_MPP_ITC_IPC".MACHINE_ON_DELAYED;
END_REGION

REGION Network 20: IMMEDIATE STOP AND STOP END OF CYCLE ALARMS
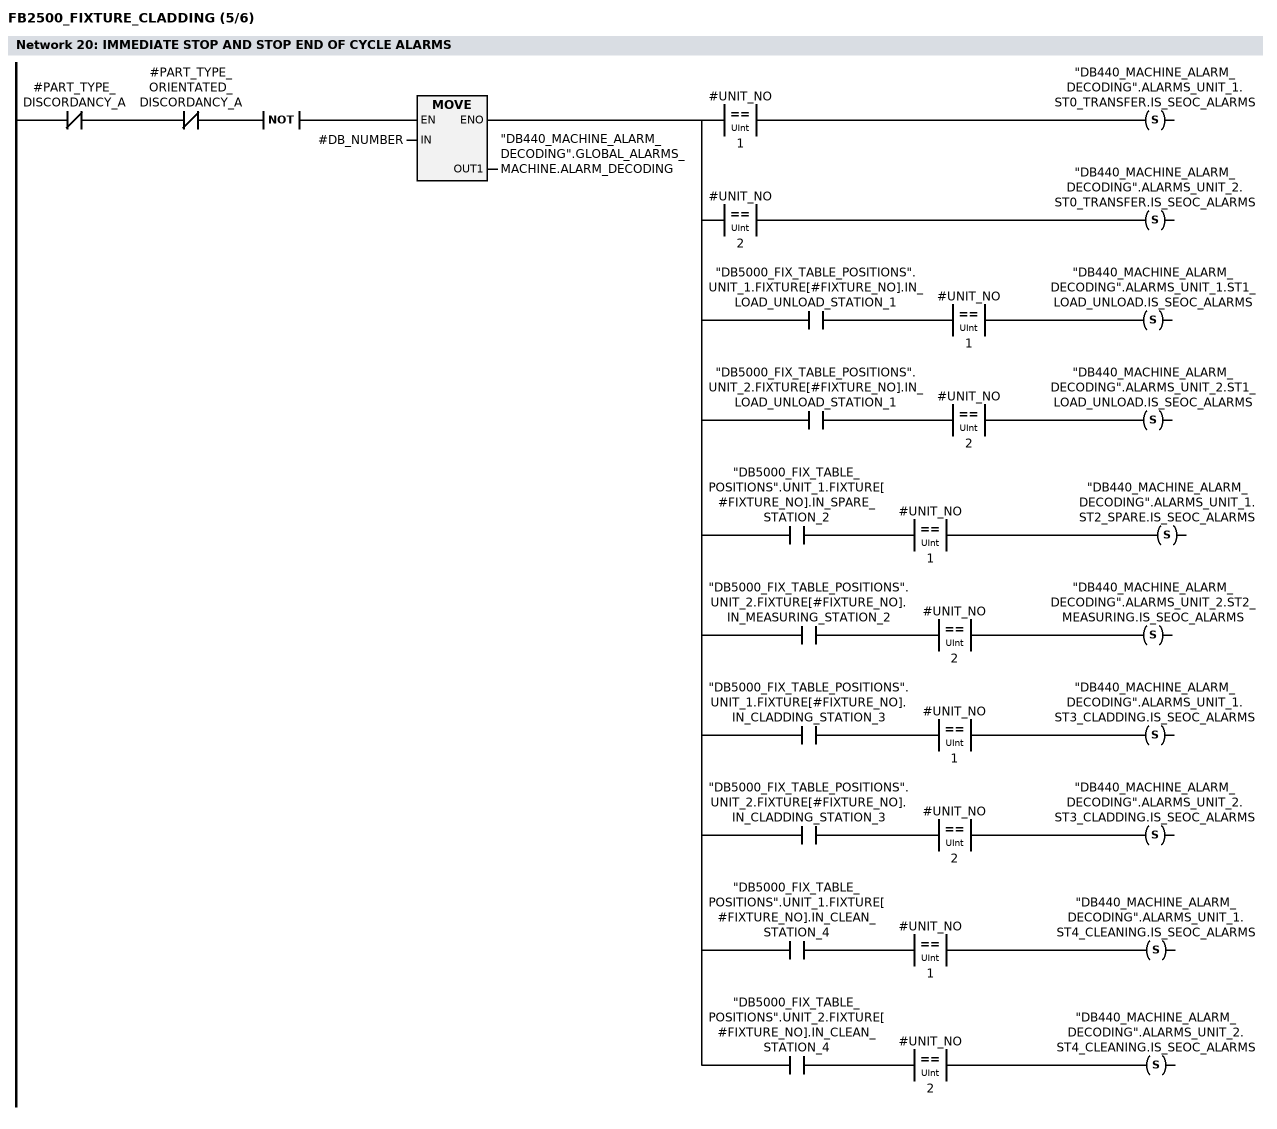
   RUNG wire#powerrail
      I_Contact( #PART_TYPE_DISCORDANCY_A )
      I_Contact( #PART_TYPE_ORIENTATED_DISCORDANCY_A )
      Not()
      Move(in := #DB_NUMBER, out1 => "DB440_MACHINE_ALARM_DECODING".GLOBAL_ALARMS_MACHINE.ALARM_DECODING)
      wire#w1
      { S7_Templates := "SrcType := UInt" } EQ_Contact(in1 := #UNIT_NO, in2 := 1)
      S_Coil( "DB440_MACHINE_ALARM_DECODING".ALARMS_UNIT_1.ST0_TRANSFER.IS_SEOC_ALARMS )
   END_RUNG
   RUNG wire#w1
      { S7_Templates := "SrcType := UInt" } EQ_Contact(in1 := #UNIT_NO, in2 := 2)
      S_Coil( "DB440_MACHINE_ALARM_DECODING".ALARMS_UNIT_2.ST0_TRANSFER.IS_SEOC_ALARMS )
   END_RUNG
   RUNG wire#w1
      Contact( "DB5000_FIX_TABLE_POSITIONS".UNIT_1.FIXTURE[#FIXTURE_NO].IN_LOAD_UNLOAD_STATION_1 )
      { S7_Templates := "SrcType := UInt" } EQ_Contact(in1 := #UNIT_NO, in2 := 1)
      S_Coil( "DB440_MACHINE_ALARM_DECODING".ALARMS_UNIT_1.ST1_LOAD_UNLOAD.IS_SEOC_ALARMS )
   END_RUNG
   RUNG wire#w1
      Contact( "DB5000_FIX_TABLE_POSITIONS".UNIT_2.FIXTURE[#FIXTURE_NO].IN_LOAD_UNLOAD_STATION_1 )
      { S7_Templates := "SrcType := UInt" } EQ_Contact(in1 := #UNIT_NO, in2 := 2)
      S_Coil( "DB440_MACHINE_ALARM_DECODING".ALARMS_UNIT_2.ST1_LOAD_UNLOAD.IS_SEOC_ALARMS )
   END_RUNG
   RUNG wire#w1
      Contact( "DB5000_FIX_TABLE_POSITIONS".UNIT_1.FIXTURE[#FIXTURE_NO].IN_SPARE_STATION_2 )
      { S7_Templates := "SrcType := UInt" } EQ_Contact(in1 := #UNIT_NO, in2 := 1)
      S_Coil( "DB440_MACHINE_ALARM_DECODING".ALARMS_UNIT_1.ST2_SPARE.IS_SEOC_ALARMS )
   END_RUNG
   RUNG wire#w1
      Contact( "DB5000_FIX_TABLE_POSITIONS".UNIT_2.FIXTURE[#FIXTURE_NO].IN_MEASURING_STATION_2 )
      { S7_Templates := "SrcType := UInt" } EQ_Contact(in1 := #UNIT_NO, in2 := 2)
      S_Coil( "DB440_MACHINE_ALARM_DECODING".ALARMS_UNIT_2.ST2_MEASURING.IS_SEOC_ALARMS )
   END_RUNG
   RUNG wire#w1
      Contact( "DB5000_FIX_TABLE_POSITIONS".UNIT_1.FIXTURE[#FIXTURE_NO].IN_CLADDING_STATION_3 )
      { S7_Templates := "SrcType := UInt" } EQ_Contact(in1 := #UNIT_NO, in2 := 1)
      S_Coil( "DB440_MACHINE_ALARM_DECODING".ALARMS_UNIT_1.ST3_CLADDING.IS_SEOC_ALARMS )
   END_RUNG
   RUNG wire#w1
      Contact( "DB5000_FIX_TABLE_POSITIONS".UNIT_2.FIXTURE[#FIXTURE_NO].IN_CLADDING_STATION_3 )
      { S7_Templates := "SrcType := UInt" } EQ_Contact(in1 := #UNIT_NO, in2 := 2)
      S_Coil( "DB440_MACHINE_ALARM_DECODING".ALARMS_UNIT_2.ST3_CLADDING.IS_SEOC_ALARMS )
   END_RUNG
   RUNG wire#w1
      Contact( "DB5000_FIX_TABLE_POSITIONS".UNIT_1.FIXTURE[#FIXTURE_NO].IN_CLEAN_STATION_4 )
      { S7_Templates := "SrcType := UInt" } EQ_Contact(in1 := #UNIT_NO, in2 := 1)
      S_Coil( "DB440_MACHINE_ALARM_DECODING".ALARMS_UNIT_1.ST4_CLEANING.IS_SEOC_ALARMS )
   END_RUNG
   RUNG wire#w1
      Contact( "DB5000_FIX_TABLE_POSITIONS".UNIT_2.FIXTURE[#FIXTURE_NO].IN_CLEAN_STATION_4 )
      { S7_Templates := "SrcType := UInt" } EQ_Contact(in1 := #UNIT_NO, in2 := 2)
      S_Coil( "DB440_MACHINE_ALARM_DECODING".ALARMS_UNIT_2.ST4_CLEANING.IS_SEOC_ALARMS )
   END_RUNG
   // the same network as SCL:
   #_w1 := NOT (NOT #PART_TYPE_DISCORDANCY_A AND NOT #PART_TYPE_ORIENTATED_DISCORDANCY_A);
   IF #_w1 THEN "DB440_MACHINE_ALARM_DECODING".GLOBAL_ALARMS_MACHINE.ALARM_DECODING := #DB_NUMBER; END_IF;
   IF #_w1 AND (#UNIT_NO = 1) THEN
       "DB440_MACHINE_ALARM_DECODING".ALARMS_UNIT_1.ST0_TRANSFER.IS_SEOC_ALARMS := TRUE;
   END_IF;
   IF #_w1 AND (#UNIT_NO = 2) THEN
       "DB440_MACHINE_ALARM_DECODING".ALARMS_UNIT_2.ST0_TRANSFER.IS_SEOC_ALARMS := TRUE;
   END_IF;
   IF #_w1 AND "DB5000_FIX_TABLE_POSITIONS".UNIT_1.FIXTURE[#FIXTURE_NO].IN_LOAD_UNLOAD_STATION_1 AND (#UNIT_NO = 1) THEN
       "DB440_MACHINE_ALARM_DECODING".ALARMS_UNIT_1.ST1_LOAD_UNLOAD.IS_SEOC_ALARMS := TRUE;
   END_IF;
   IF #_w1 AND "DB5000_FIX_TABLE_POSITIONS".UNIT_2.FIXTURE[#FIXTURE_NO].IN_LOAD_UNLOAD_STATION_1 AND (#UNIT_NO = 2) THEN
       "DB440_MACHINE_ALARM_DECODING".ALARMS_UNIT_2.ST1_LOAD_UNLOAD.IS_SEOC_ALARMS := TRUE;
   END_IF;
   IF #_w1 AND "DB5000_FIX_TABLE_POSITIONS".UNIT_1.FIXTURE[#FIXTURE_NO].IN_SPARE_STATION_2 AND (#UNIT_NO = 1) THEN
       "DB440_MACHINE_ALARM_DECODING".ALARMS_UNIT_1.ST2_SPARE.IS_SEOC_ALARMS := TRUE;
   END_IF;
   IF #_w1 AND "DB5000_FIX_TABLE_POSITIONS".UNIT_2.FIXTURE[#FIXTURE_NO].IN_MEASURING_STATION_2 AND (#UNIT_NO = 2) THEN
       "DB440_MACHINE_ALARM_DECODING".ALARMS_UNIT_2.ST2_MEASURING.IS_SEOC_ALARMS := TRUE;
   END_IF;
   IF #_w1 AND "DB5000_FIX_TABLE_POSITIONS".UNIT_1.FIXTURE[#FIXTURE_NO].IN_CLADDING_STATION_3 AND (#UNIT_NO = 1) THEN
       "DB440_MACHINE_ALARM_DECODING".ALARMS_UNIT_1.ST3_CLADDING.IS_SEOC_ALARMS := TRUE;
   END_IF;
   IF #_w1 AND "DB5000_FIX_TABLE_POSITIONS".UNIT_2.FIXTURE[#FIXTURE_NO].IN_CLADDING_STATION_3 AND (#UNIT_NO = 2) THEN
       "DB440_MACHINE_ALARM_DECODING".ALARMS_UNIT_2.ST3_CLADDING.IS_SEOC_ALARMS := TRUE;
   END_IF;
   IF #_w1 AND "DB5000_FIX_TABLE_POSITIONS".UNIT_1.FIXTURE[#FIXTURE_NO].IN_CLEAN_STATION_4 AND (#UNIT_NO = 1) THEN
       "DB440_MACHINE_ALARM_DECODING".ALARMS_UNIT_1.ST4_CLEANING.IS_SEOC_ALARMS := TRUE;
   END_IF;
   IF #_w1 AND "DB5000_FIX_TABLE_POSITIONS".UNIT_2.FIXTURE[#FIXTURE_NO].IN_CLEAN_STATION_4 AND (#UNIT_NO = 2) THEN
       "DB440_MACHINE_ALARM_DECODING".ALARMS_UNIT_2.ST4_CLEANING.IS_SEOC_ALARMS := TRUE;
   END_IF;
END_REGION

REGION Network 21: RETURN HOME POSITION AND STOP END OF CYCLE ALARMS
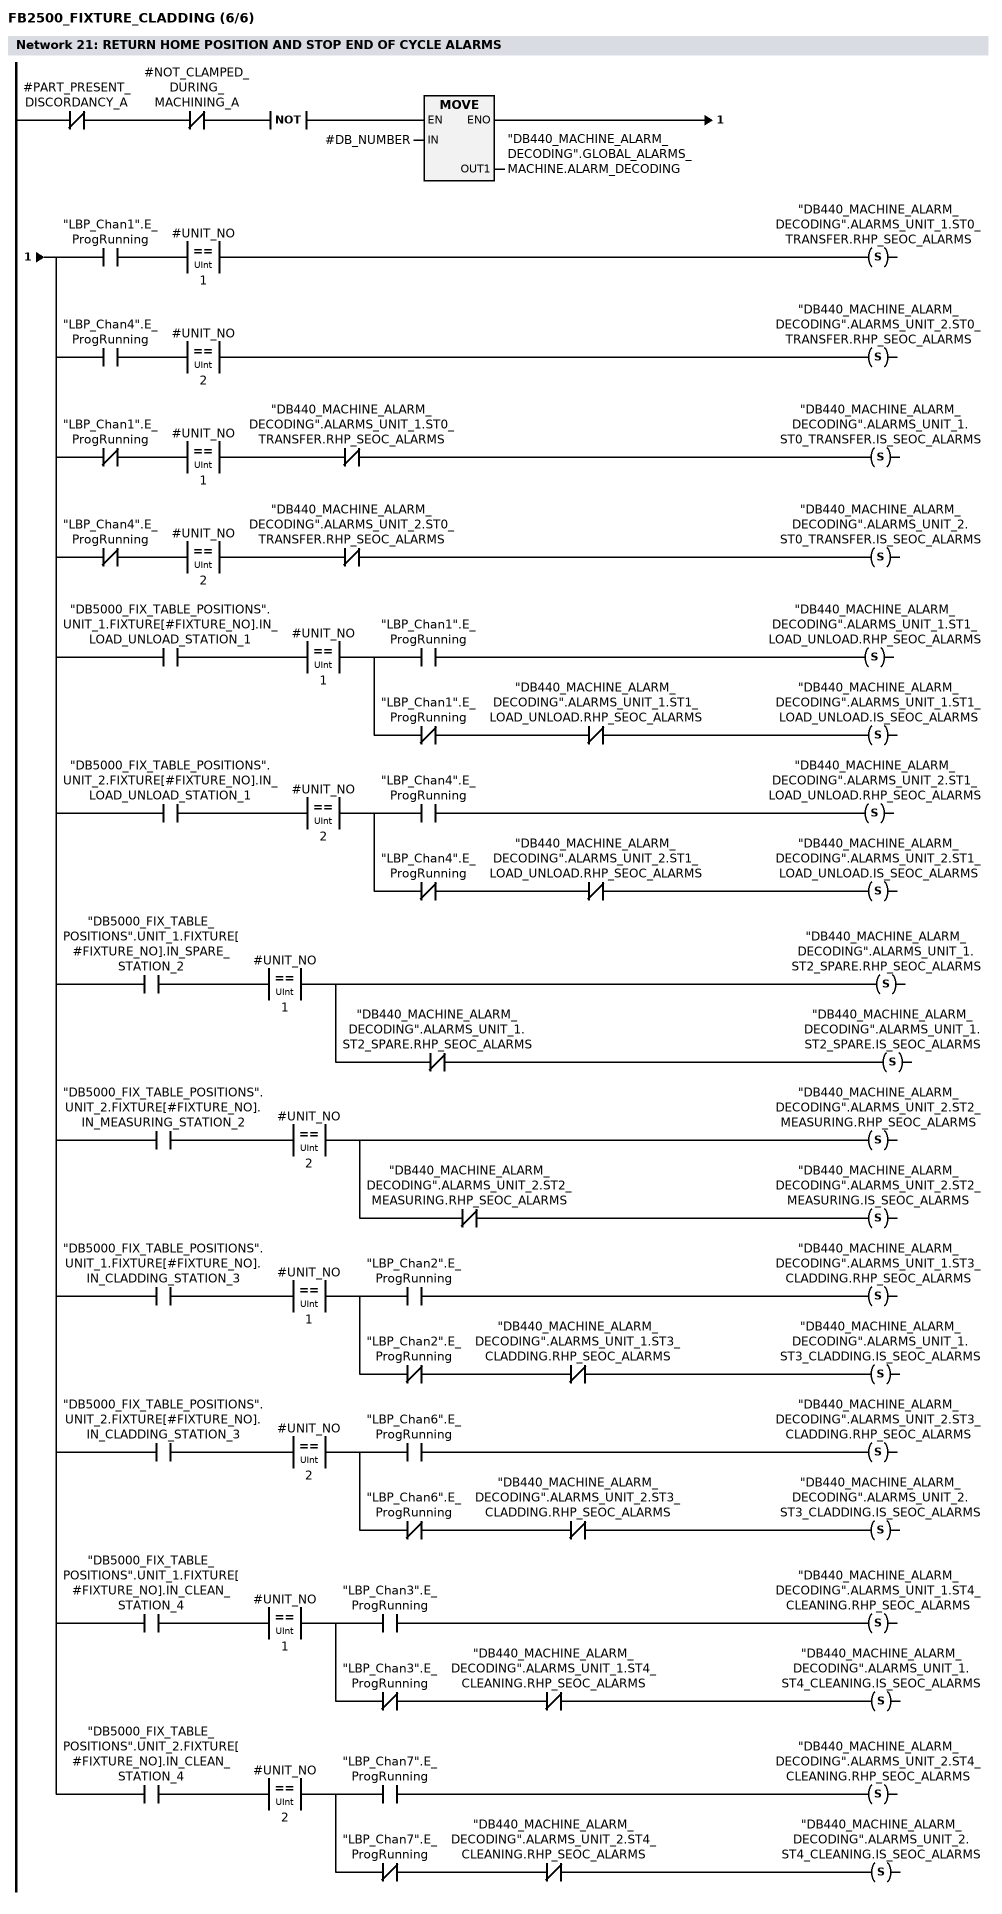
   RUNG wire#powerrail
      I_Contact( #PART_PRESENT_DISCORDANCY_A )
      I_Contact( #NOT_CLAMPED_DURING_MACHINING_A )
      Not()
      Move(in := #DB_NUMBER, out1 => "DB440_MACHINE_ALARM_DECODING".GLOBAL_ALARMS_MACHINE.ALARM_DECODING)
      wire#w1
      Contact( "LBP_Chan1".E_ProgRunning )
      { S7_Templates := "SrcType := UInt" } EQ_Contact(in1 := #UNIT_NO, in2 := 1)
      S_Coil( "DB440_MACHINE_ALARM_DECODING".ALARMS_UNIT_1.ST0_TRANSFER.RHP_SEOC_ALARMS )
   END_RUNG
   RUNG wire#w1
      Contact( "LBP_Chan4".E_ProgRunning )
      { S7_Templates := "SrcType := UInt" } EQ_Contact(in1 := #UNIT_NO, in2 := 2)
      S_Coil( "DB440_MACHINE_ALARM_DECODING".ALARMS_UNIT_2.ST0_TRANSFER.RHP_SEOC_ALARMS )
   END_RUNG
   RUNG wire#w1
      I_Contact( "LBP_Chan1".E_ProgRunning )
      { S7_Templates := "SrcType := UInt" } EQ_Contact(in1 := #UNIT_NO, in2 := 1)
      I_Contact( "DB440_MACHINE_ALARM_DECODING".ALARMS_UNIT_1.ST0_TRANSFER.RHP_SEOC_ALARMS )
      S_Coil( "DB440_MACHINE_ALARM_DECODING".ALARMS_UNIT_1.ST0_TRANSFER.IS_SEOC_ALARMS )
   END_RUNG
   RUNG wire#w1
      I_Contact( "LBP_Chan4".E_ProgRunning )
      { S7_Templates := "SrcType := UInt" } EQ_Contact(in1 := #UNIT_NO, in2 := 2)
      I_Contact( "DB440_MACHINE_ALARM_DECODING".ALARMS_UNIT_2.ST0_TRANSFER.RHP_SEOC_ALARMS )
      S_Coil( "DB440_MACHINE_ALARM_DECODING".ALARMS_UNIT_2.ST0_TRANSFER.IS_SEOC_ALARMS )
   END_RUNG
   RUNG wire#w1
      Contact( "DB5000_FIX_TABLE_POSITIONS".UNIT_1.FIXTURE[#FIXTURE_NO].IN_LOAD_UNLOAD_STATION_1 )
      { S7_Templates := "SrcType := UInt" } EQ_Contact(in1 := #UNIT_NO, in2 := 1)
      wire#w2
      Contact( "LBP_Chan1".E_ProgRunning )
      S_Coil( "DB440_MACHINE_ALARM_DECODING".ALARMS_UNIT_1.ST1_LOAD_UNLOAD.RHP_SEOC_ALARMS )
   END_RUNG
   RUNG wire#w2
      I_Contact( "LBP_Chan1".E_ProgRunning )
      I_Contact( "DB440_MACHINE_ALARM_DECODING".ALARMS_UNIT_1.ST1_LOAD_UNLOAD.RHP_SEOC_ALARMS )
      S_Coil( "DB440_MACHINE_ALARM_DECODING".ALARMS_UNIT_1.ST1_LOAD_UNLOAD.IS_SEOC_ALARMS )
   END_RUNG
   RUNG wire#w1
      Contact( "DB5000_FIX_TABLE_POSITIONS".UNIT_2.FIXTURE[#FIXTURE_NO].IN_LOAD_UNLOAD_STATION_1 )
      { S7_Templates := "SrcType := UInt" } EQ_Contact(in1 := #UNIT_NO, in2 := 2)
      wire#w3
      Contact( "LBP_Chan4".E_ProgRunning )
      S_Coil( "DB440_MACHINE_ALARM_DECODING".ALARMS_UNIT_2.ST1_LOAD_UNLOAD.RHP_SEOC_ALARMS )
   END_RUNG
   RUNG wire#w3
      I_Contact( "LBP_Chan4".E_ProgRunning )
      I_Contact( "DB440_MACHINE_ALARM_DECODING".ALARMS_UNIT_2.ST1_LOAD_UNLOAD.RHP_SEOC_ALARMS )
      S_Coil( "DB440_MACHINE_ALARM_DECODING".ALARMS_UNIT_2.ST1_LOAD_UNLOAD.IS_SEOC_ALARMS )
   END_RUNG
   RUNG wire#w1
      Contact( "DB5000_FIX_TABLE_POSITIONS".UNIT_1.FIXTURE[#FIXTURE_NO].IN_SPARE_STATION_2 )
      { S7_Templates := "SrcType := UInt" } EQ_Contact(in1 := #UNIT_NO, in2 := 1)
      wire#w4
      S_Coil( "DB440_MACHINE_ALARM_DECODING".ALARMS_UNIT_1.ST2_SPARE.RHP_SEOC_ALARMS )
   END_RUNG
   RUNG wire#w4
      I_Contact( "DB440_MACHINE_ALARM_DECODING".ALARMS_UNIT_1.ST2_SPARE.RHP_SEOC_ALARMS )
      S_Coil( "DB440_MACHINE_ALARM_DECODING".ALARMS_UNIT_1.ST2_SPARE.IS_SEOC_ALARMS )
   END_RUNG
   RUNG wire#w1
      Contact( "DB5000_FIX_TABLE_POSITIONS".UNIT_2.FIXTURE[#FIXTURE_NO].IN_MEASURING_STATION_2 )
      { S7_Templates := "SrcType := UInt" } EQ_Contact(in1 := #UNIT_NO, in2 := 2)
      wire#w5
      S_Coil( "DB440_MACHINE_ALARM_DECODING".ALARMS_UNIT_2.ST2_MEASURING.RHP_SEOC_ALARMS )
   END_RUNG
   RUNG wire#w5
      I_Contact( "DB440_MACHINE_ALARM_DECODING".ALARMS_UNIT_2.ST2_MEASURING.RHP_SEOC_ALARMS )
      S_Coil( "DB440_MACHINE_ALARM_DECODING".ALARMS_UNIT_2.ST2_MEASURING.IS_SEOC_ALARMS )
   END_RUNG
   RUNG wire#w1
      Contact( "DB5000_FIX_TABLE_POSITIONS".UNIT_1.FIXTURE[#FIXTURE_NO].IN_CLADDING_STATION_3 )
      { S7_Templates := "SrcType := UInt" } EQ_Contact(in1 := #UNIT_NO, in2 := 1)
      wire#w6
      Contact( "LBP_Chan2".E_ProgRunning )
      S_Coil( "DB440_MACHINE_ALARM_DECODING".ALARMS_UNIT_1.ST3_CLADDING.RHP_SEOC_ALARMS )
   END_RUNG
   RUNG wire#w6
      I_Contact( "LBP_Chan2".E_ProgRunning )
      I_Contact( "DB440_MACHINE_ALARM_DECODING".ALARMS_UNIT_1.ST3_CLADDING.RHP_SEOC_ALARMS )
      S_Coil( "DB440_MACHINE_ALARM_DECODING".ALARMS_UNIT_1.ST3_CLADDING.IS_SEOC_ALARMS )
   END_RUNG
   RUNG wire#w1
      Contact( "DB5000_FIX_TABLE_POSITIONS".UNIT_2.FIXTURE[#FIXTURE_NO].IN_CLADDING_STATION_3 )
      { S7_Templates := "SrcType := UInt" } EQ_Contact(in1 := #UNIT_NO, in2 := 2)
      wire#w7
      Contact( "LBP_Chan6".E_ProgRunning )
      S_Coil( "DB440_MACHINE_ALARM_DECODING".ALARMS_UNIT_2.ST3_CLADDING.RHP_SEOC_ALARMS )
   END_RUNG
   RUNG wire#w7
      I_Contact( "LBP_Chan6".E_ProgRunning )
      I_Contact( "DB440_MACHINE_ALARM_DECODING".ALARMS_UNIT_2.ST3_CLADDING.RHP_SEOC_ALARMS )
      S_Coil( "DB440_MACHINE_ALARM_DECODING".ALARMS_UNIT_2.ST3_CLADDING.IS_SEOC_ALARMS )
   END_RUNG
   RUNG wire#w1
      Contact( "DB5000_FIX_TABLE_POSITIONS".UNIT_1.FIXTURE[#FIXTURE_NO].IN_CLEAN_STATION_4 )
      { S7_Templates := "SrcType := UInt" } EQ_Contact(in1 := #UNIT_NO, in2 := 1)
      wire#w8
      Contact( "LBP_Chan3".E_ProgRunning )
      S_Coil( "DB440_MACHINE_ALARM_DECODING".ALARMS_UNIT_1.ST4_CLEANING.RHP_SEOC_ALARMS )
   END_RUNG
   RUNG wire#w8
      I_Contact( "LBP_Chan3".E_ProgRunning )
      I_Contact( "DB440_MACHINE_ALARM_DECODING".ALARMS_UNIT_1.ST4_CLEANING.RHP_SEOC_ALARMS )
      S_Coil( "DB440_MACHINE_ALARM_DECODING".ALARMS_UNIT_1.ST4_CLEANING.IS_SEOC_ALARMS )
   END_RUNG
   RUNG wire#w1
      Contact( "DB5000_FIX_TABLE_POSITIONS".UNIT_2.FIXTURE[#FIXTURE_NO].IN_CLEAN_STATION_4 )
      { S7_Templates := "SrcType := UInt" } EQ_Contact(in1 := #UNIT_NO, in2 := 2)
      wire#w9
      Contact( "LBP_Chan7".E_ProgRunning )
      S_Coil( "DB440_MACHINE_ALARM_DECODING".ALARMS_UNIT_2.ST4_CLEANING.RHP_SEOC_ALARMS )
   END_RUNG
   RUNG wire#w9
      I_Contact( "LBP_Chan7".E_ProgRunning )
      I_Contact( "DB440_MACHINE_ALARM_DECODING".ALARMS_UNIT_2.ST4_CLEANING.RHP_SEOC_ALARMS )
      S_Coil( "DB440_MACHINE_ALARM_DECODING".ALARMS_UNIT_2.ST4_CLEANING.IS_SEOC_ALARMS )
   END_RUNG
   // the same network as SCL:
   #_w1 := NOT (NOT #PART_PRESENT_DISCORDANCY_A AND NOT #NOT_CLAMPED_DURING_MACHINING_A);
   IF #_w1 THEN "DB440_MACHINE_ALARM_DECODING".GLOBAL_ALARMS_MACHINE.ALARM_DECODING := #DB_NUMBER; END_IF;
   IF #_w1 AND "LBP_Chan1".E_ProgRunning AND (#UNIT_NO = 1) THEN
       "DB440_MACHINE_ALARM_DECODING".ALARMS_UNIT_1.ST0_TRANSFER.RHP_SEOC_ALARMS := TRUE;
   END_IF;
   IF #_w1 AND "LBP_Chan4".E_ProgRunning AND (#UNIT_NO = 2) THEN
       "DB440_MACHINE_ALARM_DECODING".ALARMS_UNIT_2.ST0_TRANSFER.RHP_SEOC_ALARMS := TRUE;
   END_IF;
   IF #_w1 AND NOT "LBP_Chan1".E_ProgRunning AND (#UNIT_NO = 1) AND NOT "DB440_MACHINE_ALARM_DECODING".ALARMS_UNIT_1.ST0_TRANSFER.RHP_SEOC_ALARMS THEN
       "DB440_MACHINE_ALARM_DECODING".ALARMS_UNIT_1.ST0_TRANSFER.IS_SEOC_ALARMS := TRUE;
   END_IF;
   IF #_w1 AND NOT "LBP_Chan4".E_ProgRunning AND (#UNIT_NO = 2) AND NOT "DB440_MACHINE_ALARM_DECODING".ALARMS_UNIT_2.ST0_TRANSFER.RHP_SEOC_ALARMS THEN
       "DB440_MACHINE_ALARM_DECODING".ALARMS_UNIT_2.ST0_TRANSFER.IS_SEOC_ALARMS := TRUE;
   END_IF;
   #_w2 := #_w1 AND "DB5000_FIX_TABLE_POSITIONS".UNIT_1.FIXTURE[#FIXTURE_NO].IN_LOAD_UNLOAD_STATION_1 AND (#UNIT_NO = 1);
   IF #_w2 AND "LBP_Chan1".E_ProgRunning THEN
       "DB440_MACHINE_ALARM_DECODING".ALARMS_UNIT_1.ST1_LOAD_UNLOAD.RHP_SEOC_ALARMS := TRUE;
   END_IF;
   IF #_w2 AND NOT "LBP_Chan1".E_ProgRunning AND NOT "DB440_MACHINE_ALARM_DECODING".ALARMS_UNIT_1.ST1_LOAD_UNLOAD.RHP_SEOC_ALARMS THEN
       "DB440_MACHINE_ALARM_DECODING".ALARMS_UNIT_1.ST1_LOAD_UNLOAD.IS_SEOC_ALARMS := TRUE;
   END_IF;
   #_w3 := #_w1 AND "DB5000_FIX_TABLE_POSITIONS".UNIT_2.FIXTURE[#FIXTURE_NO].IN_LOAD_UNLOAD_STATION_1 AND (#UNIT_NO = 2);
   IF #_w3 AND "LBP_Chan4".E_ProgRunning THEN
       "DB440_MACHINE_ALARM_DECODING".ALARMS_UNIT_2.ST1_LOAD_UNLOAD.RHP_SEOC_ALARMS := TRUE;
   END_IF;
   IF #_w3 AND NOT "LBP_Chan4".E_ProgRunning AND NOT "DB440_MACHINE_ALARM_DECODING".ALARMS_UNIT_2.ST1_LOAD_UNLOAD.RHP_SEOC_ALARMS THEN
       "DB440_MACHINE_ALARM_DECODING".ALARMS_UNIT_2.ST1_LOAD_UNLOAD.IS_SEOC_ALARMS := TRUE;
   END_IF;
   #_w4 := #_w1 AND "DB5000_FIX_TABLE_POSITIONS".UNIT_1.FIXTURE[#FIXTURE_NO].IN_SPARE_STATION_2 AND (#UNIT_NO = 1);
   IF #_w4 THEN "DB440_MACHINE_ALARM_DECODING".ALARMS_UNIT_1.ST2_SPARE.RHP_SEOC_ALARMS := TRUE; END_IF;
   IF #_w4 AND NOT "DB440_MACHINE_ALARM_DECODING".ALARMS_UNIT_1.ST2_SPARE.RHP_SEOC_ALARMS THEN
       "DB440_MACHINE_ALARM_DECODING".ALARMS_UNIT_1.ST2_SPARE.IS_SEOC_ALARMS := TRUE;
   END_IF;
   #_w5 := #_w1 AND "DB5000_FIX_TABLE_POSITIONS".UNIT_2.FIXTURE[#FIXTURE_NO].IN_MEASURING_STATION_2 AND (#UNIT_NO = 2);
   IF #_w5 THEN "DB440_MACHINE_ALARM_DECODING".ALARMS_UNIT_2.ST2_MEASURING.RHP_SEOC_ALARMS := TRUE; END_IF;
   IF #_w5 AND NOT "DB440_MACHINE_ALARM_DECODING".ALARMS_UNIT_2.ST2_MEASURING.RHP_SEOC_ALARMS THEN
       "DB440_MACHINE_ALARM_DECODING".ALARMS_UNIT_2.ST2_MEASURING.IS_SEOC_ALARMS := TRUE;
   END_IF;
   #_w6 := #_w1 AND "DB5000_FIX_TABLE_POSITIONS".UNIT_1.FIXTURE[#FIXTURE_NO].IN_CLADDING_STATION_3 AND (#UNIT_NO = 1);
   IF #_w6 AND "LBP_Chan2".E_ProgRunning THEN
       "DB440_MACHINE_ALARM_DECODING".ALARMS_UNIT_1.ST3_CLADDING.RHP_SEOC_ALARMS := TRUE;
   END_IF;
   IF #_w6 AND NOT "LBP_Chan2".E_ProgRunning AND NOT "DB440_MACHINE_ALARM_DECODING".ALARMS_UNIT_1.ST3_CLADDING.RHP_SEOC_ALARMS THEN
       "DB440_MACHINE_ALARM_DECODING".ALARMS_UNIT_1.ST3_CLADDING.IS_SEOC_ALARMS := TRUE;
   END_IF;
   #_w7 := #_w1 AND "DB5000_FIX_TABLE_POSITIONS".UNIT_2.FIXTURE[#FIXTURE_NO].IN_CLADDING_STATION_3 AND (#UNIT_NO = 2);
   IF #_w7 AND "LBP_Chan6".E_ProgRunning THEN
       "DB440_MACHINE_ALARM_DECODING".ALARMS_UNIT_2.ST3_CLADDING.RHP_SEOC_ALARMS := TRUE;
   END_IF;
   IF #_w7 AND NOT "LBP_Chan6".E_ProgRunning AND NOT "DB440_MACHINE_ALARM_DECODING".ALARMS_UNIT_2.ST3_CLADDING.RHP_SEOC_ALARMS THEN
       "DB440_MACHINE_ALARM_DECODING".ALARMS_UNIT_2.ST3_CLADDING.IS_SEOC_ALARMS := TRUE;
   END_IF;
   #_w8 := #_w1 AND "DB5000_FIX_TABLE_POSITIONS".UNIT_1.FIXTURE[#FIXTURE_NO].IN_CLEAN_STATION_4 AND (#UNIT_NO = 1);
   IF #_w8 AND "LBP_Chan3".E_ProgRunning THEN
       "DB440_MACHINE_ALARM_DECODING".ALARMS_UNIT_1.ST4_CLEANING.RHP_SEOC_ALARMS := TRUE;
   END_IF;
   IF #_w8 AND NOT "LBP_Chan3".E_ProgRunning AND NOT "DB440_MACHINE_ALARM_DECODING".ALARMS_UNIT_1.ST4_CLEANING.RHP_SEOC_ALARMS THEN
       "DB440_MACHINE_ALARM_DECODING".ALARMS_UNIT_1.ST4_CLEANING.IS_SEOC_ALARMS := TRUE;
   END_IF;
   #_w9 := #_w1 AND "DB5000_FIX_TABLE_POSITIONS".UNIT_2.FIXTURE[#FIXTURE_NO].IN_CLEAN_STATION_4 AND (#UNIT_NO = 2);
   IF #_w9 AND "LBP_Chan7".E_ProgRunning THEN
       "DB440_MACHINE_ALARM_DECODING".ALARMS_UNIT_2.ST4_CLEANING.RHP_SEOC_ALARMS := TRUE;
   END_IF;
   IF #_w9 AND NOT "LBP_Chan7".E_ProgRunning AND NOT "DB440_MACHINE_ALARM_DECODING".ALARMS_UNIT_2.ST4_CLEANING.RHP_SEOC_ALARMS THEN
       "DB440_MACHINE_ALARM_DECODING".ALARMS_UNIT_2.ST4_CLEANING.IS_SEOC_ALARMS := TRUE;
   END_IF;
END_REGION
END_FUNCTION_BLOCK
